// Brief: Master Arm Cart Control
FUNCTION_BLOCK PUBLIC FB_StateCtrlCart EXTENDS FB_MasterArmCtrlBase
VAR_INPUT
END_VAR
VAR_OUTPUT
END_VAR
VAR
END_VAR

METHOD PUBLIC init : BOOL
VAR_IN_OUT CONSTANT
	i_masterArm	:FB_MasterArm;
END_VAR
VAR_IN_OUT 
	r_masterArmCtrlCmd :ST_ArmCtrlCmds;
END_VAR
SUPER^.Init(i_masterArm,r_masterArmCtrlCmd);

// check if to hold the command joint position unchanged
checkToHoldLastCmds(i_masterArm,r_masterArmCtrlCmd);
END_METHOD

END_FUNCTION_BLOCK

(* stored: Version 1.1.0.1, ProductVersion 3.1.4024.12
   POU FB_StateCtrlCart: Id {acf69b98-a94c-45d6-930a-e719a9a02026}, SpecialFunc None
   Method init: Id {1dc1fdc9-dd5b-4a4c-998e-6b8ceff7fdd6} *)
